// TIA Portal project "Sorting line_Project" (V16)
// Vorlageprojekt für das Buch mit Zielsystem S7-1200

(* hardware
DEVICE "S7-1200-Station_1"  S7-1200 Station
   slot 0: "Baugruppenträger_0"  Rack  V1.0
   slot 1: "PLC_1"  CPU 1211C DC/DC/DC  6ES7 211-1AE40-0XB0  V4.1
*)

// ===== PLC "PLC_1"  CPU 1211C DC/DC/DC =====

VAR_GLOBAL   // PLC tag table "Standard-Variablentabelle"
   "xPbStart" AT %I0.1 : Bool;
   "xPbStop" AT %I0.3 : Bool;
   "xStateStart" AT %M0.0 : Bool;
   "xSensorAtExit" AT %I0.0 : Bool;
   "xPbReset" AT %I0.2 : Bool;
   "xPbStartLed" AT %Q1.1 : Bool;
   "xPbStopLed" AT %Q1.3 : Bool;
   "xPbResetLed" AT %Q1.2 : Bool;
   "xSorterBelt_1" AT %Q0.4 : Bool;
   "xSorterRotate_1" AT %Q0.3 : Bool;
   "xSorterBelt_2" AT %Q0.6 : Bool;
   "xSorterRotate_2" AT %Q0.5 : Bool;
   "xSorterBelt_3" AT %Q1.0 : Bool;
   "xSorterRotate_3" AT %Q0.7 : Bool;
   "xStoper" AT %Q0.1 : Bool;
   "xConveyorEntryMotor" AT %Q0.0 : Bool;
   "xConveyorOutputMotor" AT %Q0.2 : Bool;
   "diVisionSensor" AT %ID30 : DInt;
   "xStep_ConvSort_20_SetSorters" AT %M2.2 : Bool;
   "xStep_ConvEntry_30_MoveFurther" AT %M3.3 : Bool;
   "xMem1" AT %M0.4 : Bool;
   "xStep_ConvEntry_20_WaitForConvSort" AT %M3.2 : Bool;
   "diOrderNr" AT %MD10 : DInt;
   "xStep_ConvEntry_10_WaitForProduct" AT %M3.1 : Bool;
   "xStep_ConvEntry_0_Init" AT %M3.0 : Bool;
   "xStep_ConvSort_0_Init" AT %M2.0 : Bool;
   "xStep_ConvSort_30_ProductPushed" AT %M2.3 : Bool;
   "xStep_ConvSort_10_WaitForProducation" AT %M2.1 : Bool;
   "xMem0" AT %M0.1 : Bool;
   "System_Byte" AT %MB1 : Byte;
   "FirstScan" AT %M1.0 : Bool;
   "DiagStatusUpdate" AT %M1.1 : Bool;
   "AlwaysTRUE" AT %M1.2 : Bool;
   "AlwaysFALSE" AT %M1.3 : Bool;
   "Clock_Byte" AT %MB50 : Byte;
   "Clock_10Hz" AT %M50.0 : Bool;
   "Clock_5Hz" AT %M50.1 : Bool;
   "Clock_2.5Hz" AT %M50.2 : Bool;
   "Clock_2Hz" AT %M50.3 : Bool;
   "Clock_1.25Hz" AT %M50.4 : Bool;
   "Clock_1Hz" AT %M50.5 : Bool;
   "Clock_0.625Hz" AT %M50.6 : Bool;
   "Clock_0.5Hz" AT %M50.7 : Bool;
   "xE-Stop" AT %I0.4 : Bool;
   "diCounterProductGreen" AT %QD30 : DInt;
   "diCounterProductBlue" AT %QD34 : DInt;
   "diCounterProductMetal" AT %QD38 : DInt;
END_VAR

// folder: System blocks/Program resources

DATA_BLOCK "IEC_Timer_0_DB_1"   // DB1
{ S7_Optimized_Access := 'TRUE' }
AUTHOR : Simatic
FAMILY : IEC
NAME : IEC_TMR
VERSION : 1.0
// stored: InstanceOfName IEC_TIMER
"IEC_TIMER"
BEGIN
END_DATA_BLOCK

DATA_BLOCK "IEC_Timer_0_DB"   // DB2
{ S7_Optimized_Access := 'TRUE' }
AUTHOR : Simatic
FAMILY : IEC
NAME : IEC_TMR
VERSION : 1.0
// stored: InstanceOfName IEC_TIMER
"IEC_TIMER"
BEGIN
END_DATA_BLOCK

DATA_BLOCK "IEC_Counter_Part_1"   // DB3
{ S7_Optimized_Access := 'TRUE' }
AUTHOR : Simatic
FAMILY : IEC
NAME : CNTR
VERSION : 1.0
// stored: InstanceOfName IEC_COUNTER
"IEC_COUNTER"
BEGIN
END_DATA_BLOCK

DATA_BLOCK "IEC_Counter_Part_2"   // DB4
{ S7_Optimized_Access := 'TRUE' }
AUTHOR : Simatic
FAMILY : IEC
NAME : CNTR
VERSION : 1.0
// stored: InstanceOfName IEC_COUNTER
"IEC_COUNTER"
BEGIN
END_DATA_BLOCK

DATA_BLOCK "IEC_Counter_Part_3"   // DB5
{ S7_Optimized_Access := 'TRUE' }
AUTHOR : Simatic
FAMILY : IEC
NAME : CNTR
VERSION : 1.0
// stored: InstanceOfName IEC_COUNTER
"IEC_COUNTER"
BEGIN
END_DATA_BLOCK

// folder: (top level)

FUNCTION "MHJ-PLC-Lab-Function-S71200" : Void   // FC9000, SCL
{ S7_Optimized_Access := 'TRUE' }
VERSION : 0.1
   VAR_TEMP
      rdTimeReturn : Int;
      outputTime : DTL;
      SyncVal : Byte;
      forVal : Int;
      forVal_2 : Int;
      Value : Byte;
   END_VAR
   VAR CONSTANT
      CompVal : Byte := 16#34;
      Value_01 : Byte := 16#11;
      Value_01_DW : DWord := 16#A165_D992;
      Value_02_DW : DWord := 16#58BE_4401;
   END_VAR
BEGIN

   #Value:=PEEK(area := 16#82,
        dbNumber := 0,
        byteOffset := 511);
   #Value := #Value + 1;

   POKE(area := 16#82,
        dbNumber := 0,
        byteOffset := 511,
        value := #Value);

   POKE(area:=16#81,
        dbNumber:=0,
        byteOffset:=1016,
        value:=#Value_01_DW);
   POKE(area := 16#81,
        dbNumber := 0,
        byteOffset := 1020,
        value := #Value_02_DW);

   POKE(area := 16#81,
        dbNumber := 0,
        byteOffset := 511,
        value := B#16#00);

   FOR #forVal := 0 TO 120 DO
       FOR #forVal_2:=0 TO 10 DO
           #rdTimeReturn:=RD_SYS_T(#outputTime);
           #rdTimeReturn := WR_SYS_T(#outputTime);
           #rdTimeReturn := RD_SYS_T(#outputTime);
           #rdTimeReturn := WR_SYS_T(#outputTime);
       END_FOR;
       #SyncVal:= PEEK(area := 16#81,
                      dbNumber := 0,
                      byteOffset := 511);
       IF #SyncVal = #CompVal THEN
          GOTO M_1;
       END_IF;
   END_FOR;
   RETURN;

   M_1:
   POKE(area := 16#81,
        dbNumber := 0,
        byteOffset := 511,
        value := B#16#0);
END_FUNCTION

ORGANIZATION_BLOCK "Main"   // OB1, LAD, ProgramCycle
TITLE = "Main Program Sweep (Cycle)"
{ S7_Optimized_Access := 'TRUE' }
VERSION : 0.1
   VAR_INPUT
      Initial_Call : Bool;   // Initial call of this OB
      Remanence : Bool;   // =True, if remanent data are available
   END_VAR
   VAR_TEMP   // added for the SCL form of the ladder/FBD networks
      _w1 : Bool;
      _w2 : Bool;
   END_VAR
BEGIN

REGION Network 1: Start/Stop system
   // Start/Stop system
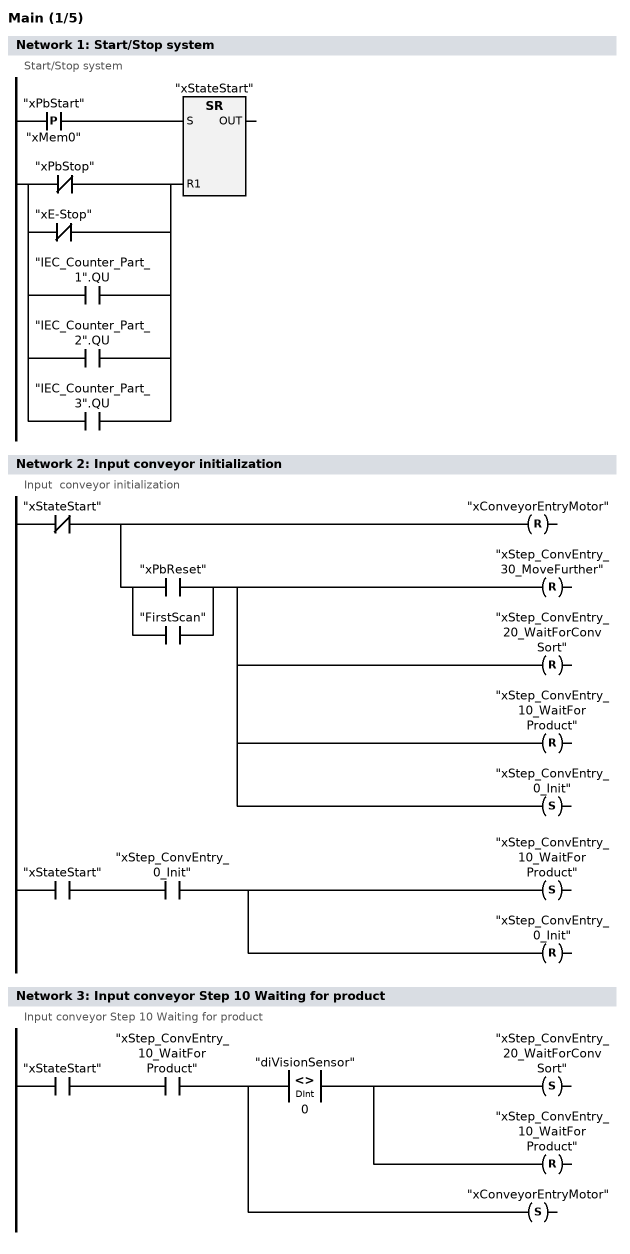
   RUNG wire#powerrail
      P_Contact(operand := "xPbStart", bit := "xMem0")
      S_SR(operand := "xStateStart", r1 := wire#w1)
   END_RUNG
   RUNG wire#powerrail
      I_Contact( "xPbStop" )
   END_RUNG wire#w1
   RUNG wire#powerrail
      I_Contact( "xE-Stop" )
   END_RUNG wire#w1
   RUNG wire#powerrail
      Contact( "IEC_Counter_Part_1".QU )
   END_RUNG wire#w1
   RUNG wire#powerrail
      Contact( "IEC_Counter_Part_2".QU )
   END_RUNG wire#w1
   RUNG wire#powerrail
      Contact( "IEC_Counter_Part_3".QU )
   END_RUNG wire#w1
   // the same network as SCL:
   #_w1 := "xPbStart" AND NOT "xMem0";   // rising edge of "xPbStart"
   "xMem0" := "xPbStart";
   IF #_w1 THEN
       "xStateStart" := TRUE;   // SR flip-flop
   END_IF;
   IF NOT "xPbStop" OR NOT "xE-Stop" OR "IEC_Counter_Part_1".QU OR "IEC_Counter_Part_2".QU OR "IEC_Counter_Part_3".QU THEN
       "xStateStart" := FALSE;
   END_IF;
END_REGION

REGION Network 2: Input conveyor initialization
   // Input  conveyor initialization
   RUNG wire#powerrail
      I_Contact( "xStateStart" )
      wire#w1
      R_Coil( "xConveyorEntryMotor" )
   END_RUNG
   RUNG wire#w1
      Contact( "xPbReset" )
      wire#w2
      R_Coil( "xStep_ConvEntry_30_MoveFurther" )
   END_RUNG
   RUNG wire#w1
      Contact( "FirstScan" )
   END_RUNG wire#w2
   RUNG wire#w2
      R_Coil( "xStep_ConvEntry_20_WaitForConvSort" )
   END_RUNG
   RUNG wire#w2
      R_Coil( "xStep_ConvEntry_10_WaitForProduct" )
   END_RUNG
   RUNG wire#w2
      S_Coil( "xStep_ConvEntry_0_Init" )
   END_RUNG
   RUNG wire#powerrail
      Contact( "xStateStart" )
      Contact( "xStep_ConvEntry_0_Init" )
      wire#w3
      S_Coil( "xStep_ConvEntry_10_WaitForProduct" )
   END_RUNG
   RUNG wire#w3
      R_Coil( "xStep_ConvEntry_0_Init" )
   END_RUNG
   // the same network as SCL:
   IF NOT "xStateStart" THEN "xConveyorEntryMotor" := FALSE; END_IF;
   IF NOT "xStateStart" AND ("xPbReset" OR "FirstScan") THEN
       "xStep_ConvEntry_30_MoveFurther" := FALSE;
       "xStep_ConvEntry_20_WaitForConvSort" := FALSE;
       "xStep_ConvEntry_10_WaitForProduct" := FALSE;
       "xStep_ConvEntry_0_Init" := TRUE;
   END_IF;
   IF "xStateStart" AND "xStep_ConvEntry_0_Init" THEN
       "xStep_ConvEntry_10_WaitForProduct" := TRUE;
       "xStep_ConvEntry_0_Init" := FALSE;
   END_IF;
END_REGION

REGION Network 3: Input conveyor Step 10 Waiting for product
   // Input conveyor Step 10 Waiting for product
   RUNG wire#powerrail
      Contact( "xStateStart" )
      Contact( "xStep_ConvEntry_10_WaitForProduct" )
      wire#w1
      { S7_Templates := "SrcType := DInt" } NE_Contact(in1 := "diVisionSensor", in2 := 0)
      wire#w2
      S_Coil( "xStep_ConvEntry_20_WaitForConvSort" )
   END_RUNG
   RUNG wire#w2
      R_Coil( "xStep_ConvEntry_10_WaitForProduct" )
   END_RUNG
   RUNG wire#w1
      S_Coil( "xConveyorEntryMotor" )
   END_RUNG
   // the same network as SCL:
   #_w1 := "xStateStart" AND "xStep_ConvEntry_10_WaitForProduct";
   IF #_w1 AND ("diVisionSensor" <> 0) THEN
       "xStep_ConvEntry_20_WaitForConvSort" := TRUE;
       "xStep_ConvEntry_10_WaitForProduct" := FALSE;
   END_IF;
   IF #_w1 THEN "xConveyorEntryMotor" := TRUE; END_IF;
END_REGION

REGION Network 4: Input conveyor Step 20 Waiting for sorting conveyor
   // Input conveyor Step 20 Waiting for sorting conveyor
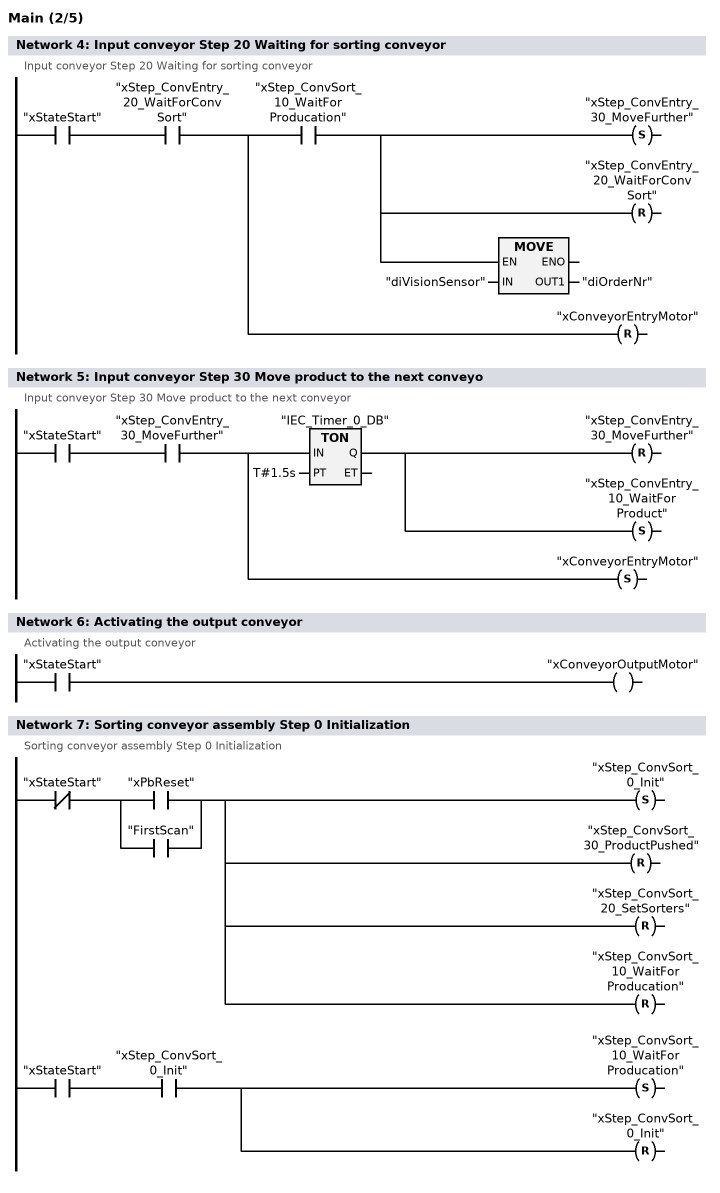
   RUNG wire#powerrail
      Contact( "xStateStart" )
      Contact( "xStep_ConvEntry_20_WaitForConvSort" )
      wire#w1
      Contact( "xStep_ConvSort_10_WaitForProducation" )
      wire#w2
      S_Coil( "xStep_ConvEntry_30_MoveFurther" )
   END_RUNG
   RUNG wire#w2
      R_Coil( "xStep_ConvEntry_20_WaitForConvSort" )
   END_RUNG
   RUNG wire#w2
      Move(in := "diVisionSensor", out1 => "diOrderNr")
   END_RUNG
   RUNG wire#w1
      R_Coil( "xConveyorEntryMotor" )
   END_RUNG
   // the same network as SCL:
   #_w1 := "xStateStart" AND "xStep_ConvEntry_20_WaitForConvSort";
   IF #_w1 AND "xStep_ConvSort_10_WaitForProducation" THEN
       "xStep_ConvEntry_30_MoveFurther" := TRUE;
       "xStep_ConvEntry_20_WaitForConvSort" := FALSE;
       "diOrderNr" := "diVisionSensor";
   END_IF;
   IF #_w1 THEN "xConveyorEntryMotor" := FALSE; END_IF;
END_REGION

REGION Network 5: Input conveyor Step 30 Move product to the next conveyo
   // Input conveyor Step 30 Move product to the next conveyor
   #_w1 := "xStateStart" AND "xStep_ConvEntry_30_MoveFurther";
   "IEC_Timer_0_DB".TON(IN := #_w1, PT := T#1.5s);
   IF "IEC_Timer_0_DB".Q THEN
       "xStep_ConvEntry_30_MoveFurther" := FALSE;
       "xStep_ConvEntry_10_WaitForProduct" := TRUE;
   END_IF;
   IF #_w1 THEN "xConveyorEntryMotor" := TRUE; END_IF;
END_REGION

REGION Network 6: Activating the output conveyor
   // Activating the output conveyor
   RUNG wire#powerrail
      Contact( "xStateStart" )
      Coil( "xConveyorOutputMotor" )
   END_RUNG
   // the same network as SCL:
   "xConveyorOutputMotor" := "xStateStart";
END_REGION

REGION Network 7: Sorting conveyor assembly Step 0 Initialization
   // Sorting conveyor assembly Step 0 Initialization
   RUNG wire#powerrail
      I_Contact( "xStateStart" )
      wire#w1
      Contact( "xPbReset" )
      wire#w2
      S_Coil( "xStep_ConvSort_0_Init" )
   END_RUNG
   RUNG wire#w1
      Contact( "FirstScan" )
   END_RUNG wire#w2
   RUNG wire#w2
      R_Coil( "xStep_ConvSort_30_ProductPushed" )
   END_RUNG
   RUNG wire#w2
      R_Coil( "xStep_ConvSort_20_SetSorters" )
   END_RUNG
   RUNG wire#w2
      R_Coil( "xStep_ConvSort_10_WaitForProducation" )
   END_RUNG
   RUNG wire#powerrail
      Contact( "xStateStart" )
      Contact( "xStep_ConvSort_0_Init" )
      wire#w3
      S_Coil( "xStep_ConvSort_10_WaitForProducation" )
   END_RUNG
   RUNG wire#w3
      R_Coil( "xStep_ConvSort_0_Init" )
   END_RUNG
   // the same network as SCL:
   IF NOT "xStateStart" AND ("xPbReset" OR "FirstScan") THEN
       "xStep_ConvSort_0_Init" := TRUE;
       "xStep_ConvSort_30_ProductPushed" := FALSE;
       "xStep_ConvSort_20_SetSorters" := FALSE;
       "xStep_ConvSort_10_WaitForProducation" := FALSE;
   END_IF;
   IF "xStateStart" AND "xStep_ConvSort_0_Init" THEN
       "xStep_ConvSort_10_WaitForProducation" := TRUE;
       "xStep_ConvSort_0_Init" := FALSE;
   END_IF;
END_REGION

REGION Network 8: Sorting conveyor assembly Step 10 Waiting for the input conveyor to provide the product
   // Sorting conveyor assembly Step 10 Waiting for the input conveyor to provide the product
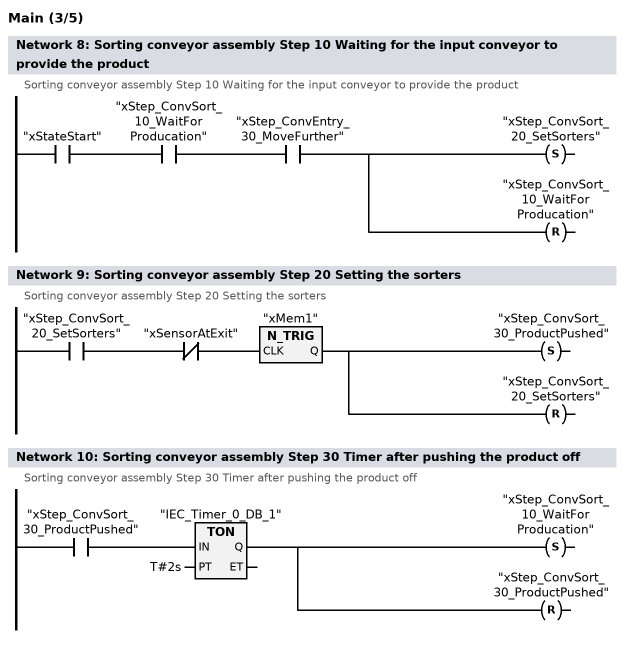
   RUNG wire#powerrail
      Contact( "xStateStart" )
      Contact( "xStep_ConvSort_10_WaitForProducation" )
      Contact( "xStep_ConvEntry_30_MoveFurther" )
      wire#w1
      S_Coil( "xStep_ConvSort_20_SetSorters" )
   END_RUNG
   RUNG wire#w1
      R_Coil( "xStep_ConvSort_10_WaitForProducation" )
   END_RUNG
   // the same network as SCL:
   IF "xStateStart" AND "xStep_ConvSort_10_WaitForProducation" AND "xStep_ConvEntry_30_MoveFurther" THEN
       "xStep_ConvSort_20_SetSorters" := TRUE;
       "xStep_ConvSort_10_WaitForProducation" := FALSE;
   END_IF;
END_REGION

REGION Network 9: Sorting conveyor assembly Step 20 Setting the sorters
   // Sorting conveyor assembly Step 20 Setting the sorters
   RUNG wire#powerrail
      Contact( "xStep_ConvSort_20_SetSorters" )
      I_Contact( "xSensorAtExit" )
      N_Trig( "xMem1" )
      wire#w1
      S_Coil( "xStep_ConvSort_30_ProductPushed" )
   END_RUNG
   RUNG wire#w1
      R_Coil( "xStep_ConvSort_20_SetSorters" )
   END_RUNG
   // the same network as SCL:
   #_w1 := "xStep_ConvSort_20_SetSorters" AND NOT "xSensorAtExit";
   #_w2 := NOT #_w1 AND "xMem1";   // falling edge
   "xMem1" := #_w1;
   IF #_w2 THEN
       "xStep_ConvSort_30_ProductPushed" := TRUE;
       "xStep_ConvSort_20_SetSorters" := FALSE;
   END_IF;
END_REGION

REGION Network 10: Sorting conveyor assembly Step 30 Timer after pushing the product off
   // Sorting conveyor assembly Step 30 Timer after pushing the product off
   "IEC_Timer_0_DB_1".TON(IN := "xStep_ConvSort_30_ProductPushed", PT := T#2s);
   IF "IEC_Timer_0_DB_1".Q THEN
       "xStep_ConvSort_10_WaitForProducation" := TRUE;
       "xStep_ConvSort_30_ProductPushed" := FALSE;
   END_IF;
END_REGION

REGION Network 11: Checking if the elements fall within the given range
   // checking if the elements fall within the given range
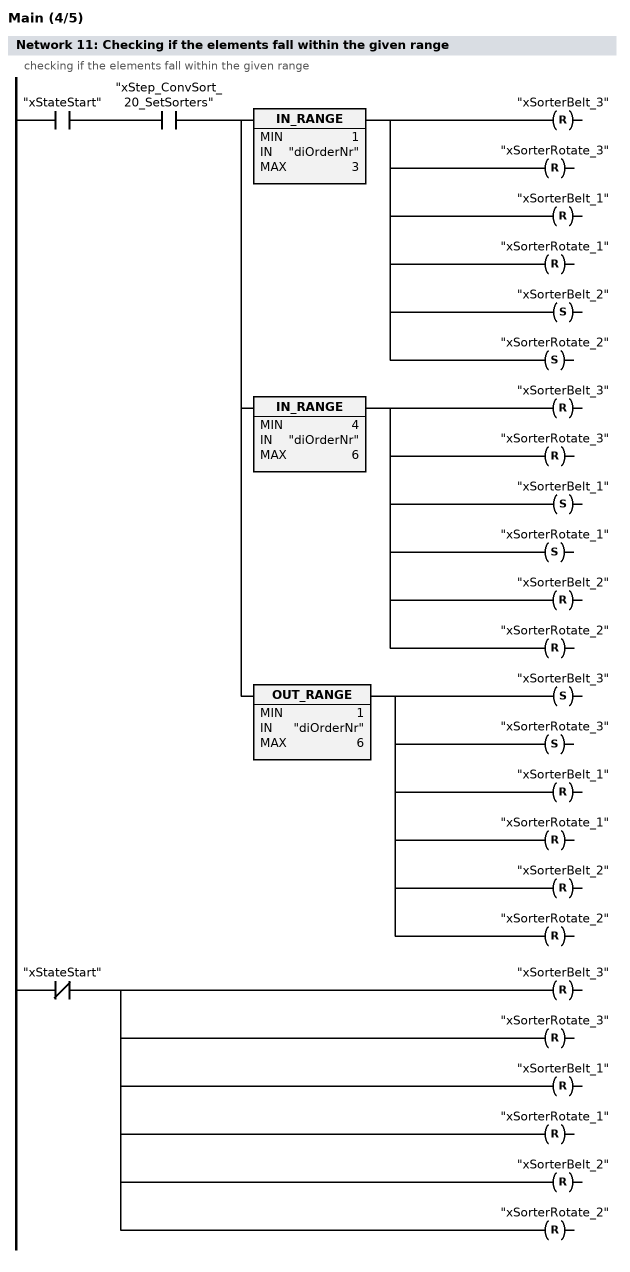
   #_w1 := "xStateStart" AND "xStep_ConvSort_20_SetSorters";
   IF #_w1 AND (1 <= "diOrderNr") AND ("diOrderNr" <= 3) THEN
       "xSorterBelt_3" := FALSE;
       "xSorterRotate_3" := FALSE;
       "xSorterBelt_1" := FALSE;
       "xSorterRotate_1" := FALSE;
       "xSorterBelt_2" := TRUE;
       "xSorterRotate_2" := TRUE;
   END_IF;
   IF #_w1 AND (4 <= "diOrderNr") AND ("diOrderNr" <= 6) THEN
       "xSorterBelt_3" := FALSE;
       "xSorterRotate_3" := FALSE;
       "xSorterBelt_1" := TRUE;
       "xSorterRotate_1" := TRUE;
       "xSorterBelt_2" := FALSE;
       "xSorterRotate_2" := FALSE;
   END_IF;
   IF #_w1 AND (("diOrderNr" < 1) OR ("diOrderNr" > 6)) THEN
       "xSorterBelt_3" := TRUE;
       "xSorterRotate_3" := TRUE;
       "xSorterBelt_1" := FALSE;
       "xSorterRotate_1" := FALSE;
       "xSorterBelt_2" := FALSE;
       "xSorterRotate_2" := FALSE;
   END_IF;
   IF NOT "xStateStart" THEN
       "xSorterBelt_3" := FALSE;
       "xSorterRotate_3" := FALSE;
       "xSorterBelt_1" := FALSE;
       "xSorterRotate_1" := FALSE;
       "xSorterBelt_2" := FALSE;
       "xSorterRotate_2" := FALSE;
   END_IF;
END_REGION

REGION Network 12: Push buton's LEDs
   // Push buton's LEDs
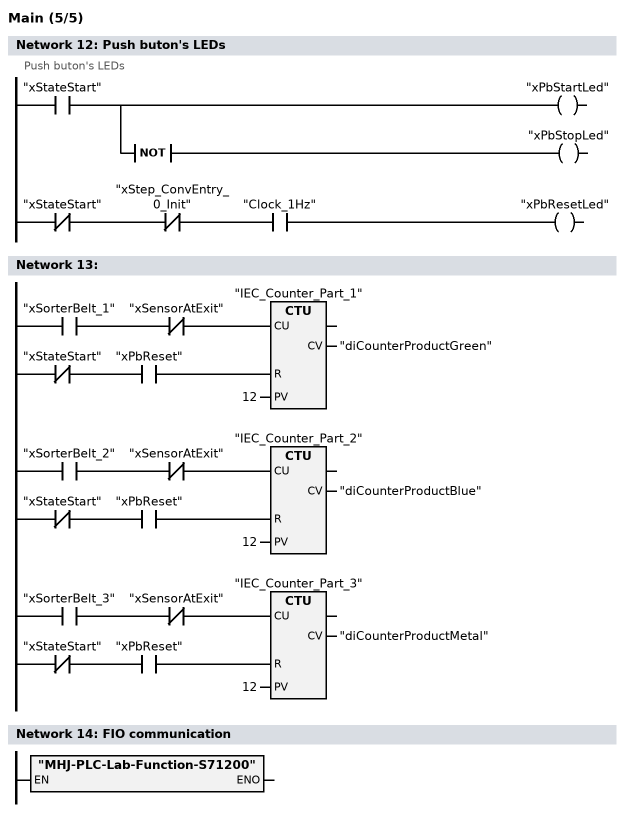
   RUNG wire#powerrail
      Contact( "xStateStart" )
      wire#w1
      Coil( "xPbStartLed" )
   END_RUNG
   RUNG wire#w1
      Not()
      Coil( "xPbStopLed" )
   END_RUNG
   RUNG wire#powerrail
      I_Contact( "xStateStart" )
      I_Contact( "xStep_ConvEntry_0_Init" )
      Contact( "Clock_1Hz" )
      Coil( "xPbResetLed" )
   END_RUNG
   // the same network as SCL:
   "xPbStartLed" := "xStateStart";
   "xPbStopLed" := NOT "xStateStart";
   "xPbResetLed" := NOT "xStateStart" AND NOT "xStep_ConvEntry_0_Init" AND "Clock_1Hz";
END_REGION

REGION Network 13
   "IEC_Counter_Part_1".CTU(CU := "xSorterBelt_1" AND NOT "xSensorAtExit",
                           R := NOT "xStateStart" AND "xPbReset",
                           PV := 12,
                           CV => "diCounterProductGreen");
   "IEC_Counter_Part_2".CTU(CU := "xSorterBelt_2" AND NOT "xSensorAtExit",
                           R := NOT "xStateStart" AND "xPbReset",
                           PV := 12,
                           CV => "diCounterProductBlue");
   "IEC_Counter_Part_3".CTU(CU := "xSorterBelt_3" AND NOT "xSensorAtExit",
                           R := NOT "xStateStart" AND "xPbReset",
                           PV := 12,
                           CV => "diCounterProductMetal");
END_REGION

REGION Network 14: FIO communication
   RUNG wire#powerrail
      "MHJ-PLC-Lab-Function-S71200"()
   END_RUNG
   // the same network as SCL:
   "MHJ-PLC-Lab-Function-S71200"();
END_REGION
END_ORGANIZATION_BLOCK